TYPE EL5151_ENC_Outputs :
STRUCT
	{attribute addProperty Name "Control"}
	Control AT %Q* : EL5101_Control;
	{attribute addProperty Name "Set counter value"}
	SetCounterValue AT %Q* : UINT;
END_STRUCT
END_TYPE

(* stored: Version 1.1.0.1, ProductVersion 3.1.4024.9
   DUT EL5151_ENC_Outputs: Id {d7d17bcf-b44d-011a-1d6d-a2dae9c0466c} *)
